// TIA Portal V17 export
// export: Created 2022-02-03T14:45:10.7908853Z, ExportSetting WithDefaults, DisplayName Totally Integrated Automation Portal, DisplayVersion V17, DisplayName TIA Portal Openness, DisplayVersion V17, DisplayName TIA Portal Version Control Interface, DisplayVersion V17, DisplayName SINAMICS Startdrive Advanced, DisplayVersion V17, DisplayName SINAMICS Startdrive G130, G150, S120, S150, SINAMICS MV, S210, DisplayVersion V17, DisplayName SINAMICS Startdrive G110M, G120, G120C, G120D, G120P, G115D, DisplayVersion V17, DisplayName STEP 7 Professional, DisplayVersion V17, DisplayName STEP 7 Safety, DisplayVersion V17, DisplayName WinCC Advanced, DisplayVersion V17
FUNCTION "Fault" : Void   // FC4, LAD
VERSION : 0.1
// stored: Access Published, AutoNumber true, IsIECCheckEnabled false, SetENOAutomatically false, UDAEnableTagReadback false
   VAR_INPUT
      conveyorAutoLeft : Bool;   // Conveyor drive in the left side in the automatic mode
      maxTime : Time;   // max. transport time
      acknowledgeFault : Bool;   // Acknowledge fault
   END_VAR
   VAR_IN_OUT
      conveyorFault : Bool;
      instIECTimer : TON_TIME;
   END_VAR
BEGIN

REGION Network 1
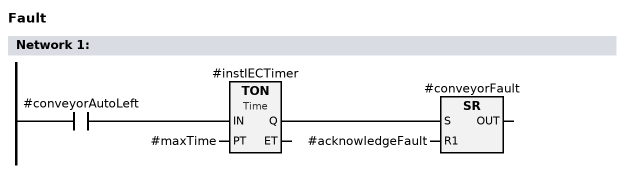
   RUNG wire#powerrail
      Contact( #conveyorAutoLeft )
      { S7_Templates := "time_type := Time" } #instIECTimer.TON(pt := #maxTime, et =>)
      S_SR(operand := #conveyorFault, r1 := #acknowledgeFault)
   END_RUNG
   // the same network as SCL:
   #instIECTimer(IN := #conveyorAutoLeft, PT := #maxTime);   // TON
   IF #instIECTimer.Q THEN
       #conveyorFault := TRUE;   // SR flip-flop
   END_IF;
   IF #acknowledgeFault THEN #conveyorFault := FALSE; END_IF;
END_REGION
END_FUNCTION
